{attribute addProperty BoxType "EL2521-0000-1016"}
{attribute addProperty Id "Set_counterAT %Q*BOOL813Set_counter_valueAT %Q*UINT16217"}
{attribute addProperty CRC "2413720468"}
{attribute addProperty SizeInBites "24"}
{attribute addProperty SizeInBytes "3"}
TYPE ENC_Control_compact_8FDE7394 :
STRUCT
	{attribute addProperty Name "Set_counter"}
	Set_counter AT %Q* : BOOL;
	{attribute addProperty Name "Set_counter_value"}
	Set_counter_value AT %Q* : UINT;
END_STRUCT
END_TYPE

(* stored: Version 1.2.0.0, ProductVersion 3.1.4024.9
   DUT ENC_Control_compact_8FDE7394: Id {507d8f21-abba-4863-b831-39da252c05a8} *)
